{attribute 'GeneratedUsingTerminal: EL6021-0000-0016'}
{attribute addProperty BoxType "EL6021-0000-0016"}
{attribute addProperty Id "EtcSlaveTerminalBaseCOM_InputsAT %I*COM_Inputs_3801C95E30COM_OutputsAT %Q*COM_Outputs_DEF408EC27WcStateAT %I*WcState_9091E0EB2InfoDataAT %I*InfoData_32EB74EA10"}
{attribute addProperty CRC "1283405116"}
{attribute addProperty Size "69"}
TYPE EL6021_4C7F353C EXTENDS EtcSlaveTerminalBase :
STRUCT
	{attribute addProperty Name "COM_Inputs"}
	COM_Inputs : COM_Inputs_3801C95E;
	{attribute addProperty Name "COM_Outputs"}
	COM_Outputs : COM_Outputs_DEF408EC;
	{attribute addProperty Name "WcState"}
	WcState : WcState_9091E0EB;
	{attribute addProperty Name "InfoData"}
	InfoData : InfoData_32EB74EA;
END_STRUCT
END_TYPE

(* stored: Version 1.2.0.0, ProductVersion 3.1.4024.9
   DUT EL6021_4C7F353C: Id {5d7a7f31-778f-4662-bfe3-98918d0834c8} *)
